# EPICS StreamDevice protocol: Stream/shutter.proto
terminator = CR LF;

id {
	ExtraInput = Ignore;
	out "ID?";
	in "%39c";
}

pos {

	out "SER:POS %d";
	in "%d";
}

  debug{
	ExtraInput = Ignore;
	out "%s";
	in "%39c";
}
